// TIA Portal V16 export
// export: Created 2022-02-28T20:48:06.2133134Z, ExportSetting WithDefaults, DisplayName Totally Integrated Automation Portal, DisplayVersion V16, DisplayName TIA Portal Version Control Interface, DisplayVersion V16, DisplayName TIA Portal Openness, DisplayVersion V16, DisplayName STEP 7 Professional, DisplayVersion V16, DisplayName STEP 7 Safety, DisplayVersion V16, DisplayName WinCC Advanced, DisplayVersion V16
TYPE "UDT_DatosProd"
// stored: IsFailsafeCompliant false
   STRUCT
      Entradas : Struct
         Longitud : Int;
         Insercion : Bool;
         Dato_In : String;
         Dato_Clr : String;
         Reset : Bool;
         Extraccion : Bool;
      END_STRUCT;
      Salidas : Struct
         Dato_Out : String;
         Add_Dn : Bool;
         Ext_Dn : Bool;
      END_STRUCT;
      Buffer : Array[0..10] of String;
      valor_Camara : String;
   END_STRUCT;
END_TYPE
